DATA_BLOCK "DB_Motor_Transfer_1"
{ S7_Optimized_Access := 'TRUE' }
VERSION : 0.1
NON_RETAIN
   VAR
      Enable : Bool := TRUE;
      CmdRun : Bool := FALSE;
      FbRun : Bool := FALSE;
      OutRun : Bool := FALSE;
      Fault : Bool := FALSE;
      tStartTimeout : Time := T#2S;
   END_VAR
BEGIN
END_DATA_BLOCK
